Fanuc KAREL source: delete_me.kl

PROGRAM MyProgram
----------------------------------------------------
-- Creation date: 2020-05-25 12:20:20
-- Created by:
----------------------------------------------------
-- Version: 0.0.0.0 - 00
----------------------------------------------------
-- Function:
----------------------------------------------------
-- Last modified: 2020.05.25
-- Last modified by:
----------------------------------------------------
%COMMENT = '0.0.0.0 - 00'
%ALPHABETIZE
--%NOABORT = ERROR+COMMAND+TPENABLE
%NOPAUSE = ERROR+COMMAND+TPENABLE
%NOPAUSESHFT
%NOLOCKGROUP
%NOBUSYLAMP
--%CMOSVARS
--%CMOS2SHADOW
%SHADOWVARS
%INCLUDE KLEVKEYS
%INCLUDE KLEVKMSK
%INCLUDE KLEVCCDF
%INCLUDE KLIOUOP
%INCLUDE KLIOTYPS
----------------------------------------------------
-- CONTANTS AND TYPES
----------------------------------------------------
--CONST
--TYPE
----------------------------------------------------
-- VARIABLES
----------------------------------------------------
--VAR
----------------------------------------------------
-- ROUTINES
----------------------------------------------------
----------------------------------------------------
-- BEGIN MyProgram
----------------------------------------------------
BEGIN
    WRITE('Hello World.')
END MyProgram
